FUNCTION_BLOCK PUBLIC AutomaticControl
VAR_INPUT
    Switch: BOOL;
END_VAR
VAR
    State: INT := 0;
    ExecutingRecipe1: BOOL := FALSE;
    ExecutingRecipe2: BOOL := FALSE;
    myRecipe2: Recipe2; // Removed invalid initialization
    Tmp: BOOL;
    RestorePreviousAutomaticState: RestorePreviousAutomaticState;
END_VAR
VAR_OUTPUT
    Output: BOOL := TRUE;
END_VAR

// TwinCAT ensures that all POUs, including your AutomaticControl program 
// and Recipe1() Function Block, are executed once per cycle.

IF NOT IO.Initialized THEN
	Initialize();
	
ELSIF IO.SwitchedToAutomatic THEN
    RestorePreviousAutomaticState();
ELSE
	CountCurrentPosition();
	//Safety();
    IF IO.ButtonUpperLeft OR ExecutingRecipe1 THEN
        ExecutingRecipe1 := TRUE;
		Recipe1();
        ExecutingRecipe1 := NOT Recipe1.SuccesfullyEnded; // Update ExecutingRecipe1 based on output
    ELSIF NOT ExecutingRecipe1 AND (IO.ButtonUpperRight OR ExecutingRecipe2) THEN
        ExecutingRecipe2 := TRUE;
        myRecipe2.ExecutingRecipe2 := ExecutingRecipe2; // Pass input to the function block
        //myRecipe2(); // Call the function block
        ExecutingRecipe2 := NOT myRecipe2.SuccesfullyEnded; // Update ExecutingRecipe2 based on output
    END_IF
END_IF


// for debugging purposes:
IF IO.ButtonRed THEN
	IO.Initialized := FALSE;
END_IF

RETURN;

END_FUNCTION_BLOCK

(* stored: Version 1.1.0.1, ProductVersion 3.1.4024.13
   POU AutomaticControl: Id {f9244839-88dd-4f0f-95ab-d4274120fb90}, SpecialFunc None *)
